FUNCTION_BLOCK NOOP_INIT (* No-Op, also known as "no Operation" with INIT *)
  (* Standard: 61499-2 *)
  (* Version 1.0, 2026-05-05, franz *)
  PACKAGE iec61131::booleanOperators;
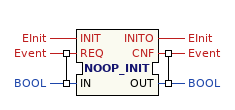
  EVENT_INPUT
    INIT : EInit; (* Initialization Request *)
    REQ WITH IN; (* Normal Execution Request *)
  END_EVENT
  EVENT_OUTPUT
    INITO : EInit; (* Initialization Confirm *)
    CNF WITH OUT; (* Execution Confirmation *)
  END_EVENT
  VAR_INPUT
    IN : BOOL; (* Input *)
  END_VAR
  VAR_OUTPUT
    OUT : BOOL; (* Output *)
  END_VAR
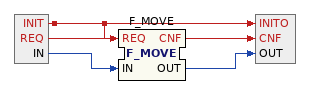
  FBS
    F_MOVE : iec61131::selection::F_MOVE; {SET_ATTRIBUTE(DataType, BOOL)}
  END_FBS
  EVENT_CONNECTIONS
    INIT TO INITO;
    REQ TO F_MOVE.REQ;
    F_MOVE.CNF TO CNF;
    INIT TO F_MOVE.REQ;
  END_CONNECTIONS
  DATA_CONNECTIONS
    IN TO F_MOVE.IN;
    F_MOVE.OUT TO OUT;
  END_CONNECTIONS
END_FUNCTION_BLOCK
